SUBAPPLICATION Uebung_010b5 (* SoftKey_F1-8 auf DigitalOutput_Q1-8 *)
  (* Standard: 61499-2; Description: Copyright (c) 2023 Meisterschulen am Ostbahnhof This program and the accompanying materials are made available under the terms of the Eclipse Public License 2.0 which is available at https://www.eclipse.org/legal/epl-2.0/ SPDX-License-Identifier: EPL-2.0 *)
  (* Version 1.0, 2023-10-23, Franz Höpfinger, Meisterschulen am Ostbahnhof *)
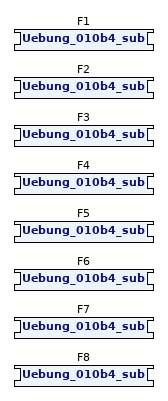
  SUBAPPS
    F1 : Uebung_010b4_sub;
    F2 : Uebung_010b4_sub;
    F3 : Uebung_010b4_sub;
    F4 : Uebung_010b4_sub;
    F5 : Uebung_010b4_sub;
    F6 : Uebung_010b4_sub;
    F7 : Uebung_010b4_sub;
    F8 : Uebung_010b4_sub;
  END_SUBAPPS
END_SUBAPPLICATION
